FUNCTION_BLOCK FB_K_Auto
VAR_INPUT
	Zasilanie:bool;
	Start:BOOL;
	Stop:BOOL;
	Pauza:BOOL;
	W_Wys:BOOL;
	W_Cof:BOOL;
	Docisk_Wys:BOOL;
	Docisk_Cof:BOOL;
	K1_Wys:BOOL;
	K1_Cof:BOOL;
	K2_Wys:BOOL;
	K2_Cof:BOOL;
	K_Dluga_Wyp:BOOL;
	K_Dluga_Cof:BOOL;
	S_Ready:BOOL;
	S_Run:BOOL;
	S_Done:BOOL;
	kolejny: BOOL;
	Safety1 : BOOL;
	Safety2  : BOOL;
	Pred_zad_podjazd: LREAL;
	Pred_zad_odjazd: LREAL;
	Reset: BOOL;
	xKartonWydany :BOOL;
	
END_VAR
VAR_OUTPUT
	S_KL_Dl:BOOL;
	S_KL1_K:BOOL;
	S_KL2_K:BOOL;
	S_Wy:BOOL;
	S_EXE:BOOL;	
	S_Docisk:BOOL;
	F2_Run:BOOL;	
	Pomp_V:BOOL;
	Pozycja:LREAL;
	Predkosc:LREAL;
	F2_CZ:INT;
	Error_ind: BOOL;
	Error_numb: INT;
	xKartonZabrany:BOOL;
	xWydajKarton:BOOL;
	
	
END_VAR
VAR
	Seq :INT;
	Czas :ARRAY[0..100] OF TON;
	CZ :TON;
	przeliczenie :INT;
	alarm_int : INT:=3;
	
END_VAR

CASE seq OF
	

0:(**)
	S_KL_Dl:=FALSE;
	S_KL1_K:=FALSE;
	S_KL2_K:=FALSE;
	S_Wy:=FALSE;
	S_EXE:=FALSE;
	S_Docisk:=FALSE;
	F2_Run:=FALSE;
	Pomp_V:=FALSE;
	F2_CZ:=0;
	
	xKartonZabrany:=FALSE;

	IF start=TRUE AND Safety1=TRUE AND Safety2=TRUE AND Zasilanie=TRUE THEN
		
	Seq:=5;

	END_IF
	

4:(*start kolejnego cyklu *)

	
	S_KL_Dl:=FALSE;
	S_KL1_K:=FALSE;
	S_KL2_K:=FALSE;
	S_Wy:=FALSE;
	S_EXE:=FALSE;
	S_Docisk:=FALSE;
	//F2_Run:=FALSE;
	Pomp_V:=FALSE;
	//F2_CZ:=0;
	
	IF kolejny=TRUE THEN
		
	Seq:=5;

	END_IF

5:(**)
	
	IF W_Cof=TRUE AND Docisk_Cof=TRUE AND K1_Cof=TRUE AND K2_Cof=TRUE AND K_Dluga_Cof=TRUE AND S_Ready=TRUE  THEN
		
	F2_CZ:=2000;
	F2_Run:=TRUE;

	Seq:=10;
	END_IF


10:(**)
	Predkosc:=Pred_zad_podjazd;		/// 900
	Pozycja:=600;
	
	IF S_Ready=TRUE THEN
	
		S_EXE:=TRUE;
	
	END_IF
	
	IF S_Run=TRUE THEN
		S_EXE:=FALSE;
		Seq:=15;
	
	END_IF

15:(**)
	IF S_Done=TRUE THEN
		Pomp_V:=TRUE;    // czy został zamontowany czujnik podcisnienie???
		xWydajKarton:=TRUE;
		
		Seq:=17; 
	END_IF
17:(**)	
		//IF GVL_IO.Vacuostat=TRUE THEN
	//	IF Czas[11].q=TRUE THEN 
		Seq:=20; 
		//END_IF
		//END_IF



20:(**)
	Pozycja:=225-((GVL_Recipe.szer_kartonu)/2);//dla malego kartonu bylo 156 //dla kartonu 370x370 was 40 
	Predkosc:=Pred_zad_odjazd;
	IF czas[0].Q=TRUE AND S_Ready=TRUE AND xKartonWydany=TRUE THEN
		xWydajKarton:=FALSE;	
	 S_EXE:=TRUE;
	 
	
	END_IF

	IF S_Run=TRUE THEN 

	Seq:=25;
	
	END_IF

25:(**)
	IF S_Done=TRUE THEN
		S_EXE:=FALSE;
		S_Docisk:=TRUE;
		xKartonZabrany:=TRUE;
		seq:=30;
	
	END_IF

30:(**)
	
	IF 	Docisk_Wys=TRUE THEN 
		xKartonZabrany:=FALSE;
	S_KL1_K:=TRUE;
	S_KL2_K:=TRUE;
		seq:=35;
	END_IF
	

35:(**)
	IF K1_Wys=TRUE AND K2_Wys=TRUE THEN
		S_KL_Dl:=TRUE;
		
		seq:=40;
	END_IF
40:(**)

	IF K_Dluga_Wyp=TRUE AND Czas[1].Q=TRUE THEN
		Pomp_V:=FALSE;
		seq:=42;
	END_IF
	
42:
	Pozycja:=225-((GVL_Recipe.szer_kartonu)/2)-20;//dla malego kartonu bylo 156 //dla kartonu 370x370 was 40
	Predkosc:=800; /// predkosc odjazdu do home
	IF  S_Ready=TRUE AND S_Run=FALSE THEN
		
	 S_EXE:=TRUE;
	 
	
	END_IF

	IF S_Run=TRUE THEN 
		
	Seq:=44;
	
	END_IF
44:
	IF S_Done=TRUE THEN
		S_Wy:=TRUE;
		Seq:=45;
	END_IF
	

45:(**)
	IF W_Wys=TRUE AND Czas[2].Q=TRUE  THEN
		
		S_KL_Dl:=FALSE;
		S_KL1_K:=FALSE;
		S_KL2_K:=FALSE;
		S_Wy:=FALSE;
		
		
		seq:=50;
	END_IF

50:(**)
	IF  W_Cof=TRUE  AND K1_Cof=TRUE AND K2_Cof=TRUE AND K_Dluga_Cof=TRUE THEN
		
	S_Docisk:=FALSE;
	seq:=4;
	END_IF

1000:(**)// Errors
	
	Error_ind:=TRUE;
	F2_Run:=FALSE;
	Pomp_V:=FALSE;  
	IF Reset=TRUE THEN
		Error_ind:=FALSE;
		Error_numb:=0;
		alarm_int:=3;
		seq:=0;
	END_IF

END_CASE

Czas[0](IN:=seq=20, PT:=T#450MS);
Czas[1](IN:=seq=40, PT:=T#0.5S);
Czas[2](IN:=seq=45, PT:=T#0.5S);

//czasowki do bledow
Czas[3](IN:=seq=5, PT:=T#5S); //Błąd gotowości do pracy
//Czas[4](IN:=seq=15, PT:=T#5S);
Czas[5](IN:=seq=25, PT:=T#5S); // Nie osiągnięto pozycji składania kartonu
Czas[6](IN:=seq=30, PT:=T#5S); // Docisk się nie wysunął
Czas[7](IN:=seq=35, PT:=T#5S); // Błąd klap
Czas[8](IN:=seq=40, PT:=T#5S); // Błąd wypychacz
Czas[9](IN:=seq=44, PT:=T#5S); // Błąd pozycji oczekiwania
Czas[10](IN:=seq=50, PT:=T#5S); // Błąd kończenia cyklu... kartoniarka nie przechodzi do stanu początkowego
Czas[11](IN:=GVL_IO.K1K3=TRUE, PT:=T#1S); // Błąd kończenia cyklu... kartoniarka nie przechodzi do stanu początkowego
// Obsługa błędów

IF Reset= FALSE THEN
FOR alarm_int:=3 TO 10 DO 
IF Czas[alarm_int].Q=TRUE THEN
	Error_numb:=alarm_int+100; // DLA KART. +100 DLA ZAKLEJARKI +200 ITD
	seq:=1000;
END_IF	
END_FOR
END_IF

IF stop=TRUE OR Safety1=FALSE OR Safety2=FALSE OR Zasilanie=FALSE  THEN 
	
	seq:=0;
		F2_Run:=FALSE;
		

	

END_IF

END_FUNCTION_BLOCK

(* stored: Version 1.1.0.1, ProductVersion 3.1.4022.12
   POU FB_K_Auto: Id {a3c4118e-c96f-4ad5-a626-dc0fe0322678}, SpecialFunc None *)
